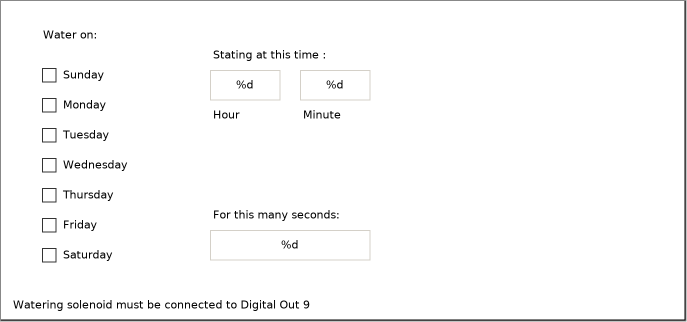
VISUALIZATION Watering  // 687x322
    Rectangle (0,0 685x320)
    Checkbox (40,60 150x30), "Sunday", variable: GVL.wateringDays[0]
    Checkbox (40,90 150x30), "Monday", variable: GVL.wateringDays[1]
    Checkbox (40,120 150x30), "Tuesday", variable: GVL.wateringDays[2]
    Checkbox (40,150 150x30), "Wednesday", variable: GVL.wateringDays[3]
    Checkbox (40,180 150x30), "Thursday", variable: GVL.wateringDays[4]
    Checkbox (40,210 150x30), "Friday", variable: GVL.wateringDays[5]
    Checkbox (40,240 150x30), "Saturday", variable: GVL.wateringDays[6]
    Textfield (210,70 70x30), "%d", text variable: GVL.HMIWateringStartHour
        OnMouseClick: write the text variable via VisuDialogs.Numpad, min 0, max 23, title 'Hour 0-23'
    Textfield (300,70 70x30), "%d", text variable: GVL.HMIWateringStartMinute
        OnMouseClick: write the text variable via VisuDialogs.Numpad, min 0, max 59, title 'Minute 0-59'
    Textfield (210,230 160x30), "%d", text variable: GVL.HMIWateringTimeSeconds
        OnMouseClick: write the text variable via VisuDialogs.Numpad, min 0, max 86400, title 'Duration (seconds)'
    Label (40,20 60x30), "Water on:"
    Label (210,40 180x30), "Stating at this time :"
    Label (210,200 140x30), "For this many seconds:"
    Label (210,100 40x30), "Hour"
    Label (300,100 80x30), "Minute"
    Label (10,290 320x30), "Watering solenoid must be connected to Digital Out 9"
END_VISUALIZATION

(* stored: Version 1.1.0.1, ProductVersion 3.1.4022.18
   Visu Watering: Id {24194610-e7ea-4b3e-b8b7-621dc9f44fe7} *)
